FUNCTION_BLOCK MyOwnContent EXTENDS TcoCore.TcoInputDialogContentContainer
VAR_INPUT
END_VAR
VAR_OUTPUT
END_VAR
VAR
    {attribute addProperty Name "<#Recipe#>"}
    Recipe : STRING;
    {attribute addProperty Name "<#Qantity#>"}
    RequiredQuantity : INT;
    {attribute addProperty Name "<#Timeout#>"}
    Timeout : DATE_AND_TIME;
    {attribute addProperty Name "<#Exclude#>"}
    Exclude : BOOL;
END_VAR

END_FUNCTION_BLOCK

(* stored: Version 1.1.0.1
   POU MyOwnContent: Id {ef1b443e-4024-02b7-1909-71231f869437}, SpecialFunc None *)
